// TIA Portal V20 export
TYPE "typeIntConditionHmiInterface"
// stored: Access Published, Namespace Unit1.Em0
   STRUCT
      Actuator_01 { S7_SetPoint := 'True'} : "LER_typeAxisActuatorCondition";   // AnodeNgBoxLockUpDown
      Actuator_02 { S7_SetPoint := 'True'} : "LER_typeAxisActuatorCondition";   // AnodeMaintenanceMovingFixFrontFwdBwd
      Actuator_03 { S7_SetPoint := 'True'} : "LER_typeAxisActuatorCondition";   // AnodeMaintenanceMovingFixFrontFwdBwd
      Actuator_04 { S7_SetPoint := 'True'} : "LER_typeAxisActuatorCondition";   // AnodeNgBoxLockUpDown
      Actuator_05 { S7_SetPoint := 'True'} : "LER_typeAxisActuatorCondition";   // AnodeMaintenanceMovingFixFrontFwdBwd
      Actuator_06 { S7_SetPoint := 'True'} : "LER_typeAxisActuatorCondition";   // AnodeNgBoxLockUpDown
      Actuator_07 { S7_SetPoint := 'True'} : "LER_typeAxisActuatorCondition";   // AnodeMaintenanceMovingFixFrontFwdBwd
   END_STRUCT;
END_TYPE
